FUNCTION POU : eq2hor
VAR_INPUT
END_VAR
VAR
END_VAR

END_FUNCTION

(* stored: Version 1.1.0.1, ProductVersion 3.1.4024.12
   POU POU: Id {fb12fcb4-55f7-4d9f-9751-eaa4648ce7c7}, SpecialFunc None *)
